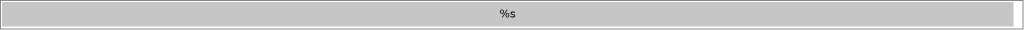
VISUALIZATION MessageRow  // 1024x30
VAR_IN_OUT
	msg:typeMessageRow;
	
	
END_VAR
    Rectangle (2,2 1011x24), "%s", text variable: msg.msgText, colour toggle: msg.isWarning, invisible if: msg.isAlarm, text list: ''
    Rectangle (2,2 1011x24), "%s", text variable: msg.msgText, colour toggle: msg.isAlarm, invisible if: msg.isWarning, text list: ''
END_VISUALIZATION

(* stored: Version 1.1.0.1, ProductVersion 3.1.4024.12
   Visu MessageRow: Id {c31f9775-5d98-4949-8bb6-dcb87c268e6f} *)
